% RSLogix 500 project TANK PUMP AND DRAIN ( ANALOG INPUT)_BAK003.RSS, saved by version 8.30.00.16 %
PROJECT "UNTITLED"    % processor: Bul.1763 MicroLogix 1100 Series B %

PROGRAM FILES
  LAD 2 "MAIN"  4 rungs
  LAD 3 "ALARMS"  7 rungs
  LAD 4 "IO"  4 rungs
  LAD 5 "CONTROLS"  6 rungs

DATA FILES
  O0 OUTPUT  5 elements
  I1 INPUT  14 elements
  S2 STATUS  66 elements
  B3 BINARY  1 elements
  T4 TIMER  4 elements
  C5 COUNTER  1 elements
  R6 CONTROL  1 elements
  N7 INTEGER  1 elements
  F8 FLOAT  1 elements

LADDER 2 "MAIN"
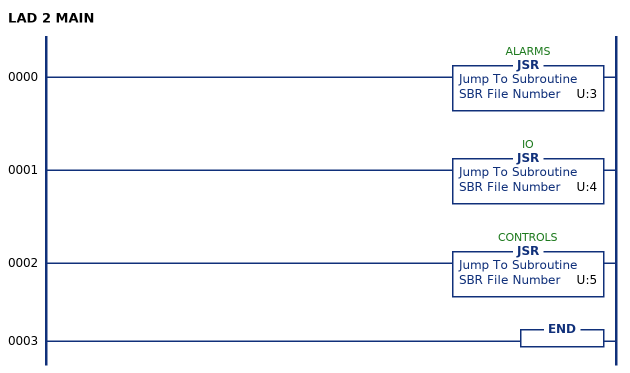
% Rung: 0 %
SOR JSR U:3 EOR
%   U:3  "ALARMS" %
% Rung: 1 %
SOR JSR U:4 EOR
%   U:4  "IO" %
% Rung: 2 %
SOR JSR U:5 EOR
%   U:5  "CONTROLS" %
% Rung: 3 %
SOR END EOR

LADDER 3 "ALARMS"
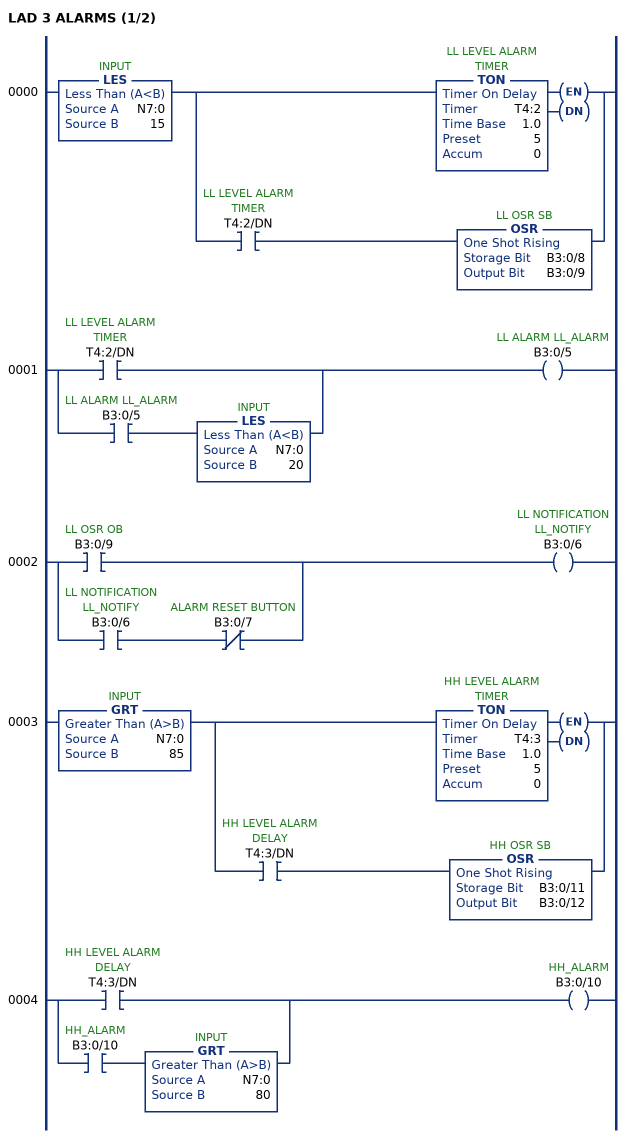
% Rung: 0 %
SOR LES N7:0 15 BST TON T4:2 1.0 5 0 NXB XIC T4:2/DN OSR B3:0/8 B3:0/9 BND EOR
%   N7:0  "INPUT" %
%   T4:2  "LL LEVEL ALARM TIMER" %
%   B3:0/8  "LL OSR SB" %
%   B3:0/9  "LL OSR OB" %
% Rung: 1 %
SOR BST XIC T4:2/DN NXB XIC B3:0/5 LES N7:0 20 BND OTE B3:0/5 EOR
%   T4:2  "LL LEVEL ALARM TIMER" %
%   B3:0/5  LL_ALARM  "LL ALARM" %
%   N7:0  "INPUT" %
% Rung: 2 %
SOR BST XIC B3:0/9 NXB XIC B3:0/6 XIO B3:0/7 BND OTE B3:0/6 EOR
%   B3:0/9  "LL OSR OB" %
%   B3:0/6  LL_NOTIFY  "LL NOTIFICATION" %
%   B3:0/7  "ALARM RESET BUTTON" %
% Rung: 3 %
SOR GRT N7:0 85 BST TON T4:3 1.0 5 0 NXB XIC T4:3/DN OSR B3:0/11 B3:0/12 BND EOR
%   N7:0  "INPUT" %
%   T4:3  "HH LEVEL ALARM TIMER" %
%   T4:3/DN  "HH LEVEL ALARM DELAY" %
%   B3:0/11  "HH OSR SB" %
%   B3:0/12  "HH OSR OB" %
% Rung: 4 %
SOR BST XIC T4:3/DN NXB XIC B3:0/10 GRT N7:0 80 BND OTE B3:0/10 EOR
%   T4:3/DN  "HH LEVEL ALARM DELAY" %
%   B3:0/10  HH_ALARM %
%   N7:0  "INPUT" %

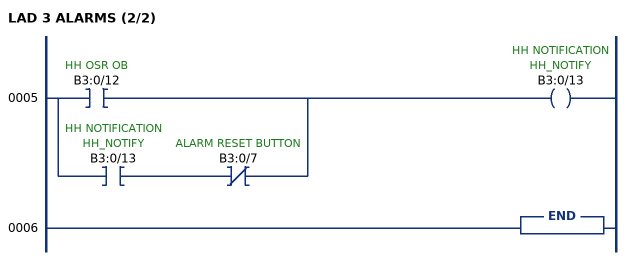
% Rung: 5 %
SOR BST XIC B3:0/12 NXB XIC B3:0/13 XIO B3:0/7 BND OTE B3:0/13 EOR
%   B3:0/12  "HH OSR OB" %
%   B3:0/13  HH_NOTIFY  "HH NOTIFICATION" %
%   B3:0/7  "ALARM RESET BUTTON" %
% Rung: 6 %
SOR END EOR

LADDER 4 "IO"
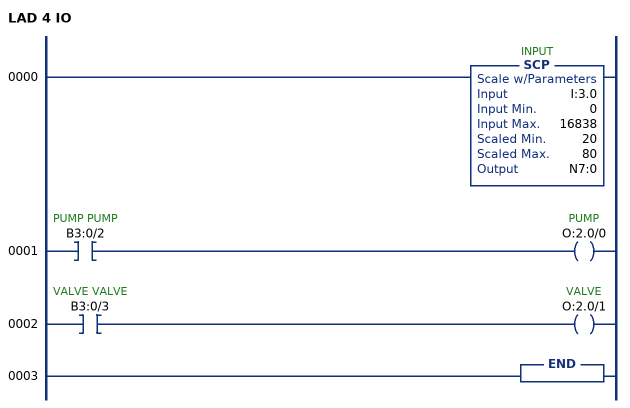
% Rung: 0 %
SOR SCP I:3.0 0 16838 20 80 N7:0 EOR
%   I:3.0  "ANALOG INPUT" %
%   N7:0  "INPUT" %
% Rung: 1 %
SOR XIC B3:0/2 OTE O:2.0/0 EOR
%   B3:0/2  PUMP  "PUMP" %
%   O:2.0/0  "PUMP" %
% Rung: 2 %
SOR XIC B3:0/3 OTE O:2.0/1 EOR
%   B3:0/3  VALVE  "VALVE" %
%   O:2.0/1  "VALVE" %
% Rung: 3 %
SOR END EOR

LADDER 5 "CONTROLS"
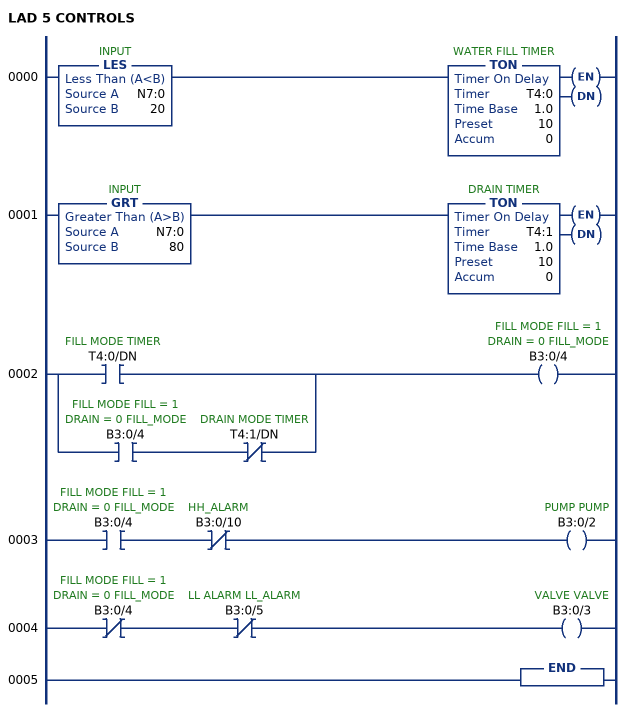
% Rung: 0 %
SOR LES N7:0 20 TON T4:0 1.0 10 0 EOR
%   N7:0  "INPUT" %
%   T4:0  "WATER FILL TIMER" %
% Rung: 1 %
SOR GRT N7:0 80 TON T4:1 1.0 10 0 EOR
%   N7:0  "INPUT" %
%   T4:1  "DRAIN TIMER" %
% Rung: 2 %
SOR BST XIC T4:0/DN NXB XIC B3:0/4 XIO T4:1/DN BND OTE B3:0/4 EOR
%   T4:0/DN  "FILL MODE TIMER" %
%   B3:0/4  FILL_MODE  "FILL MODE FILL = 1 DRAIN = 0" %
%   T4:1/DN  "DRAIN MODE TIMER" %
% Rung: 3 %
SOR XIC B3:0/4 XIO B3:0/10 OTE B3:0/2 EOR
%   B3:0/4  FILL_MODE  "FILL MODE FILL = 1 DRAIN = 0" %
%   B3:0/10  HH_ALARM %
%   B3:0/2  PUMP  "PUMP" %
% Rung: 4 %
SOR XIO B3:0/4 XIO B3:0/5 OTE B3:0/3 EOR
%   B3:0/4  FILL_MODE  "FILL MODE FILL = 1 DRAIN = 0" %
%   B3:0/5  LL_ALARM  "LL ALARM" %
%   B3:0/3  VALVE  "VALVE" %
% Rung: 5 %
SOR END EOR

OTHER DOCUMENTED ADDRESSES
  B3:0/0  "PUMP"
  B3:0/1  "VALVE"
  B3:7  ALARM_RESET  "ALARM RESET BUTTON"
  O:0.0/0  "PUMP"

REVISION NOTES
  0: ADDED ALARM AND NOTIFICATION TO LL AND HH SET POINTS

DATA TABLE (non-zero values as saved)
DATA T4
% .PRE .ACC %
% T4:0 % 10 0
% T4:1 % 10 0
% T4:2 % 5 0
% T4:3 % 5 0
